// TwinCAT 3 PLC project Abschervorrichtung
// ProgramVersion: 3.1.4026.16
// libraries:
//   Tc2_Standard, * (Beckhoff Automation GmbH)
//   Tc2_System, * (Beckhoff Automation GmbH)
// project tree:
//   DUTs/ ST_systemState.TcDUT
//   GVLs/ GVL_Abschervorrichtung.TcGVL
//   / PlcTask.TcTTO
//   POUs/ FB_Ablauf.TcPOU, FB_Betriebsarten.TcPOU, MAIN.TcPOU
// real-time tasks:
//   TASK PlcTask: cycle T#10ms, priority 20, ADS port 350

CONFIGURATION Abschervorrichtung
    RESOURCE PLC ON TwinCAT3
        TASK PlcTask(INTERVAL := T#10ms, PRIORITY := 20);
        PROGRAM MAIN WITH PlcTask : MAIN;
    END_RESOURCE
END_CONFIGURATION

// ---- DUTs/ST_systemState.TcDUT
TYPE ST_systemState :
STRUCT
	bAnlageEin: BOOL;
	bAnlageAus: BOOL;
END_STRUCT
END_TYPE

// ---- GVLs/GVL_Abschervorrichtung.TcGVL
{attribute 'qualified_only'}
VAR_GLOBAL
{region "Inputs"}
Ix_S1: BOOL; 								// Anlage Ein 
Ix_S2: BOOL; 								// Anlage Aus (Öffner) 
Ix_S3: BOOL; 								// Hand / Auto 
Ix_S4: BOOL; 								// Einzel- / Dauerzyklus 
Ix_S5: BOOL; 								// Richten 
Ix_S6: BOOL; 								// Start-Taster 
Ix_B1: BOOL; 								// Grenztaster Zyl.A eingefahren 
Ix_B2: BOOL; 								// Grenztaster Zyl.A ausgefahren 
Ix_B3: BOOL; 								// Grenztaster Zyl.B eingefahren 
Ix_B4: BOOL; 								// Grenztaster Zyl.B ausgefahren 
Ix_B5: BOOL; 								// Grenztaster Zyl.C eingefahren 
Ix_B6: BOOL; 								// Grenztaster Zyl.C ausgefahren 
Ix_B7: BOOL; 								// Grenztaster Zyl.D eingefahren 
Ix_B8: BOOL; 								// Grenztaster Zyl.D ausgefahren 	
{endregion}

{region "Outputs"}
Qx_M1: BOOL; 								// Ventil füR Zylinder A aus/einfahren 
Qx_M2: BOOL; 								// Ventil füR Zylinder B aus/einfahren 
Qx_M3: BOOL; 								// Ventil füR Zylinder C aus/einfahren 
Qx_M4: BOOL; 								// Ventil füR Zylinder D aus/einfahren 
Qx_P1: BOOL; 								// Lampe Anlage Ein 
Qx_P2: BOOL; 								// Lampe Manuelbetrieb 
Qx_P3: BOOL; 								// Lampe Autobetrieb 
Qx_P4: BOOL; 								// Lampe Dauerzyklus 
Qx_P5: BOOL; 								// Lampe STörung / NOT-Aus
{endregion}
END_VAR

// ---- POUs/MAIN.TcPOU
PROGRAM MAIN
VAR
	Ablauf: FB_Ablauf;
	Betriebsarten: FB_Betriebsarten;
END_VAR

Ablauf(stAnlagenzustand := Betriebsarten.stAnlagenzustand);
Betriebsarten();

END_PROGRAM

// ---- POUs/FB_Ablauf.TcPOU
FUNCTION_BLOCK FB_Ablauf
VAR_INPUT
	stAnlagenzustand: ST_systemState;
END_VAR
VAR_OUTPUT
END_VAR
VAR
	iStep: 			INT := 000;
END_VAR

IF stAnlagenzustand.bAnlageEin THEN
	iStep := 010;
END_IF

CASE iStep OF
	
000: 				//INIT



END_CASE

END_FUNCTION_BLOCK

// ---- POUs/FB_Betriebsarten.TcPOU
FUNCTION_BLOCK FB_Betriebsarten
VAR_INPUT
	bIStart:				BOOL;		// Starttaster 
	bIAnlageEin:			BOOL;		// Taster Anlage eingeschaltet
	bIAnlageAus: 			BOOL;		// Taster Anlage ausgeschaltet
	bIManAuto:				BOOL;		// Schalter Manuell / Automatik
	bINotAus:				BOOL;		// Not-Aus, 1 = i.O, 0 = betätigt
	bIDauerEinzel:			BOOL;		// Schalter Dauer- bzw. Einzelbetrieb, 0 = Dauer, 1 = Einzelbetrieb
END_VAR
VAR_OUTPUT
	bOAnlageEin:			BOOL;		// 1 = Anlage eingeschaltet
	bOManuell:				BOOL;		// 1 = Anlage Manuellbetrieb
	bOAuto:					BOOL;		// 1 = Anlage im Autobetrieb
	bOEinzelZyklus:			BOOL;		// 1 = Einzelzyklus aktiv
	bODauerZyklus:			BOOL;		// 1 = Dauerzyklus aktiv
	bOStoerung:				BOOL;		// 1 = Stoerung vorhanden (Not-Aus)
	bOImpEinzelSchritt:		BOOL;		// Impuls bei Einzelschrittbetrieb von Start-Taster
	bOImpDauerZyklus:		BOOL;		// Impuls bei Dauerschrittbetrieb von Start-Taster
	stAnlagenzustand:		ST_systemState;
END_VAR
VAR_IN_OUT
END_VAR
VAR
	bSVAnlageEin:			BOOL;		// Variable 1 = Anlage eingeschaltet 
	lastbEinzelImp: 		BOOL;		// Letzter Zustand Tipp-Impuls für Flankenerkennung
	lastbDauerImp: 			BOOL;		// Letzter Zustand Dauer-Impuls für Flankenerkennung
	lastbStart:				BOOL;
END_VAR

(*
- Wenn Not-Aus aktiv, alle FB-Ausgänge rücksetzen und Ausgang vqx_Störung setzen 
- vqx_AnlageEin speichernd set/reset mit vix_AnlageEin und vix_AnlageAus (Öffner) 
- Wenn Anlage nicht eigeschaltet, dann alle Ausgänge rücksetzen 
- vqx_Man wird gesetzt, wenn vix_ManAuto auf Man (False) steht und Anlage eingeschaltet ist 
- vqx_Auto wird gesetzt, wenn vix_ManAuto auf Auto (True) steht und Anlage eingeschaltet ist 
- vqx_EinzZykl wird gesetzt, wenn vix_DauerEinz auf Einzel (True) steht und die Anlage eingeschaltet ist 
- vqx_ImpEinzelSchritt wird für 1 Zyklus logisch "1" wenn der Einzel-Zyklus aktiv ist und die Anlage eingeschaltet ist und der Start-Taster gedrückt wird. 
- vqx_DauerZykl wird gesetzt, wenn vix_DauerEinz auf Dauer (False) steht und der Automatikbetrieb aktiv und die Anlage eingeschaltet ist 
- vqx_ImpDauerZykl wird für 1 Zyklus logisch "1" wenn Dauer-Zyklus aktiv ist und die Anlage eingeschaltet ist und der Start-Taster gedrückt wird.
*)

// IF bIStart THEN
// 	stAnlagenzustand.bAnlageEin := TRUE;
// END_IF

{region "not-aus"}							// If machine running and emergency stop button get hit, reset all outputs to FALSE expect output "Error"
IF bINotAus THEN			
		bOAnlageEin				:= FALSE;
		bOManuell				:= FALSE;
		bOAuto					:= FALSE;
		bOEinzelZyklus			:= FALSE;		
		bODauerZyklus			:= FALSE;
		bOImpEinzelSchritt		:= FALSE;		
		bOImpDauerZyklus		:= FALSE;
		bOStoerung				:= TRUE;
	ELSE
		bOStoerung := FALSE;
END_IF
{endregion}

{region "Anlage Ein/Aus}					// SR (reset-dominant) for status 'machine run' or 'machine isn't running'
IF bIAnlageAus THEN
	bOAnlageEin := FALSE;
ELSIF bIAnlageEin THEN
	bOAnlageEin := TRUE;
END_IF
{endregion}

{region "Anlage aus"}
IF NOT bOAnlageEin THEN
	bOAnlageEin				:= FALSE;
	bOManuell				:= FALSE;
	bOAuto					:= FALSE;
	bOEinzelZyklus			:= FALSE;		
	bODauerZyklus			:= FALSE;
	bOImpEinzelSchritt		:= FALSE;		
	bOImpDauerZyklus		:= FALSE;
	bOStoerung				:= FALSE;	
	END_IF
{endregion}
	

{region "man/auto"}
IF bOAnlageEin AND NOT bIManAuto THEN
		bOManuell 	:= TRUE;
		bOAuto 		:= FALSE;
	ELSIF bOAnlageEin AND bIManAuto THEN
		bOManuell 	:= FALSE;
		bOAuto 		:= TRUE;
	END_IF
{endregion}
	

{region "Einzelzykluis"}
IF bIDauerEinzel AND bOAnlageEin THEN
		bOEinzelZyklus := TRUE;
ELSE 
		bOEinzelZyklus := FALSE;
	END_IF
{endregion}

{region "Dauerzyklus"}
IF NOT bIDauerEinzel AND bOAuto AND bOAnlageEin THEN
		bODauerZyklus := TRUE;
	ELSE
		bODauerZyklus := FALSE;
	END_IF
{endregion}

{region "Impulse Dauer/Einzel"}
IF bOEinzelZyklus AND bOAnlageEin AND bIStart AND NOT lastbStart AND NOT lastbEinzelImp THEN
		bOImpEinzelSchritt := TRUE;
	ELSE bOImpEinzelSchritt := FALSE;
	END_IF

IF bODauerZyklus AND bOAnlageEin AND bIStart AND NOT lastbStart AND NOT lastbDauerImp THEN
		bOImpDauerZyklus := TRUE;
	ELSE bOImpDauerZyklus := FALSE;
	END_IF

lastbDauerImp 	:= bOImpDauerZyklus;
lastbEinzelImp 	:= bOImpEinzelSchritt;
lastbStart 		:= bIStart;	
{endregion}

END_FUNCTION_BLOCK
